TYPE StepTransition :
STRUCT
	actionName		: STRING;
	conditionName	: STRING;
	nextActionName	: STRING;
END_STRUCT
END_TYPE

(* stored: Version 1.1.0.1, ProductVersion 3.1.4024.11
   DUT StepTransition: Id {32049ed0-25dd-445c-a0ed-3990f8b1b9ad} *)
